// SIMATIC S7-200 project (STEP 7-Micro/WIN), CPU 224 CN REL 02.01

SYMBOL_TABLE USER1
P0_Reposo        M0.0     // Estado de espera inicial
P1_Sujecion      M0.1     // Estado de sujecion de la columna
P2_Empuje        M0.2     // Estado de entrega de la pieza inferior
P3_Retorno_E     M0.3     // Estado de retorno del cilindro de empuje
P4_Retorno_S     M0.4     // Estado de liberacion de la columna
T0_Inicio        M1.0     // Transicion Inicio Ciclo
T1_Sujeto        M1.1     // Transicion Sujecion OK
T2_Entregado     M1.2     // Transicion Entrega OK
T3_Emp_Ret       M1.3     // Transicion Empuje Retraido
T4_Suj_Ret       M1.4     // Transicion Sujecion Retraida
Ev_Marcha        M2.0     // Evento Marcha presionado y Seta OK
Ev_Pieza         M2.1     // Evento Pieza en base detectada
Ev_CilP_Ext      M2.2     // Evento Cilindro pequeno extendido
Ev_CilL_Ext      M2.3     // Evento Cilindro largo extendido
Ev_CilL_Ret      M2.4     // Evento Cilindro largo retraido
Ev_CilP_Ret      M2.5     // Evento Cilindro pequeno retraido
Ev_Pos_Pieza     M2.6     // Evento pieza en posicion
Cil_Peq_Ext      I0.0     // Sensor cilindro pequeno extendido
Cil_Peq_Ret      I0.1     // Sensor cilindro pequeno retraido
Cil_Lrg_Ext      I0.2     // Sensor cilindro largo extendido
Cil_Lrg_Ret      I0.3     // Sensor cilindro largo retraido
Pos_Pieza        I0.4     // Sensor fotoelectrico posicion pieza
Presencia_Sup    I0.5     // Sensor presencia superior
Presencia_Inf    I0.6     // Sensor presencia inferior
Sensor_Induc     I0.7     // Sensor inductivo material metalico
Btn_Marcha       I1.2     // Pulsador verde de marcha
Btn_Paro         I1.3     // Pulsador rojo de paro
Seta_Emerg       I1.4     // Zeta de emergencia (NC)
Selector_Rot     I1.5     // Selector rotatorio
V_Cil_Peq        Q0.0     // Valvula cilindro pequeno
V_Cil_Lrg        Q0.1     // Valvula cilindro largo
Lamp_Amarilla    Q0.7     // Lampara de advertencia
Lamp_Verde       Q1.0     // Lampara de marcha
Lamp_Roja        Q1.1     // Lampara de paro o falla
Sol_AP           V0.0     // Solicitud Alimentacion a Procesamiento
Ack_Sol_AP       V1.0     // Reconocimiento AP
Ack_MA           V0.1     // Reconocimiento marcha Unidad de Alimentacion
Marcha_A         V1.1     // Solicitud de marcha para la Unidad de Alimentacion
Alim_OK          V0.2     // Unidad de Alimentacion disponible
END_SYMBOL_TABLE

SYMBOL_TABLE S7-200 Symbols
First_Scan_On    SM0.1    // 仅第一个扫描周期中接通为 ON
END_SYMBOL_TABLE

ORGANIZATION_BLOCK MAIN:OB1
TITLE=UNIDAD DE ALIMENTACION - RED DE PETRI (CIPN) - 5 MODULOS (V4)
//  LOGICA BASADA EN REDES DE PETRI INTERPRETADAS
//  MODULO 1: INICIALIZACION
//  MODULO 2: EVENTOS
//  MODULO 3: DISPARO
//  MODULO 4: DINAMICA
//  MODULO 5: ACCIONES
BEGIN
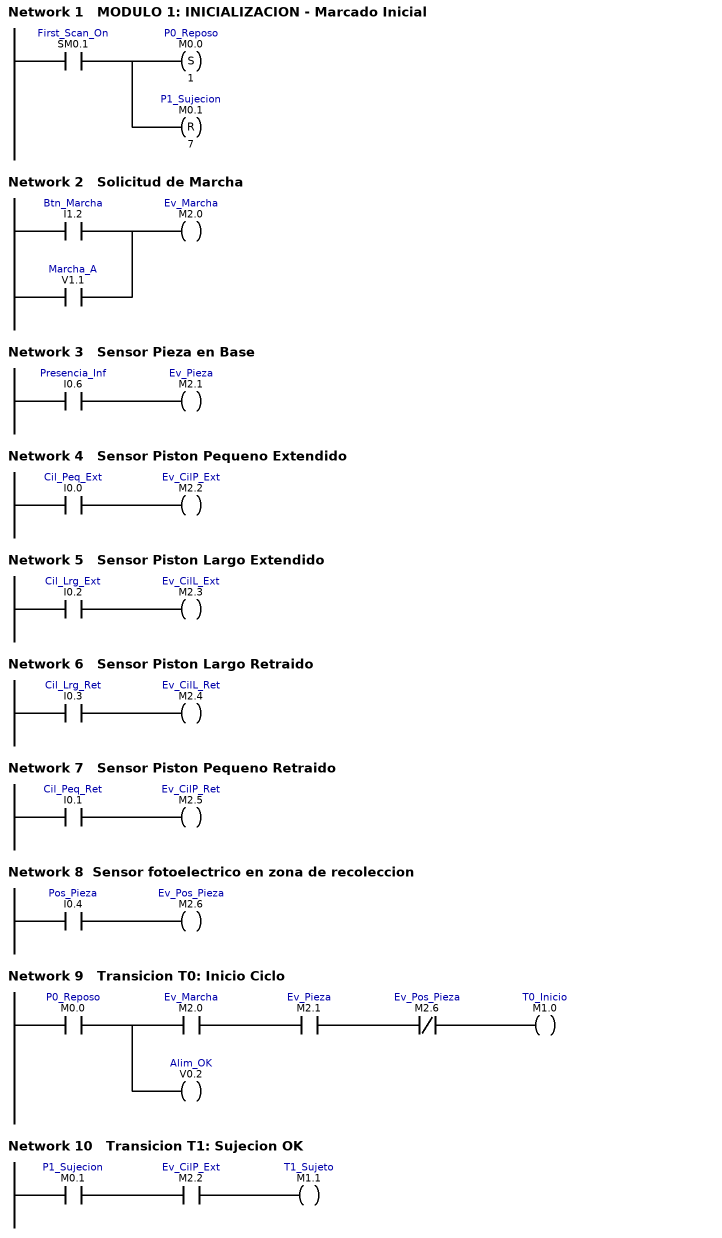
Network 1 //  MODULO 1: INICIALIZACION - Marcado Inicial
// P0 Reposo activo
// Limpieza de marcas P1-M0.7
// MODULO 2: EVENTOS (CAPTURA DE SENSORES)
LD     First_Scan_On:SM0.1
S      P0_Reposo:M0.0, 1
R      P1_Sujecion:M0.1, 7
Network 2 //  Solicitud de Marcha
LD     Btn_Marcha:I1.2
O      Marcha_A:V1.1
=      Ev_Marcha:M2.0
Network 3 //  Sensor Pieza en Base
LD     Presencia_Inf:I0.6
=      Ev_Pieza:M2.1
Network 4 //  Sensor Piston Pequeno Extendido
LD     Cil_Peq_Ext:I0.0
=      Ev_CilP_Ext:M2.2
Network 5 //  Sensor Piston Largo Extendido
LD     Cil_Lrg_Ext:I0.2
=      Ev_CilL_Ext:M2.3
Network 6 //  Sensor Piston Largo Retraido
LD     Cil_Lrg_Ret:I0.3
=      Ev_CilL_Ret:M2.4
Network 7 //  Sensor Piston Pequeno Retraido
// MODULO 3: CONDICIONES DE DISPARO (FIRING)
LD     Cil_Peq_Ret:I0.1
=      Ev_CilP_Ret:M2.5
Network 8 // Sensor fotoelectrico en zona de recoleccion
LD     Pos_Pieza:I0.4
=      Ev_Pos_Pieza:M2.6
Network 9 //  Transicion T0: Inicio Ciclo
LD     P0_Reposo:M0.0
LPS
A      Ev_Marcha:M2.0
A      Ev_Pieza:M2.1
AN     Ev_Pos_Pieza:M2.6
=      T0_Inicio:M1.0
LPP
=      Alim_OK:V0.2
Network 10 //  Transicion T1: Sujecion OK
LD     P1_Sujecion:M0.1
A      Ev_CilP_Ext:M2.2
=      T1_Sujeto:M1.1
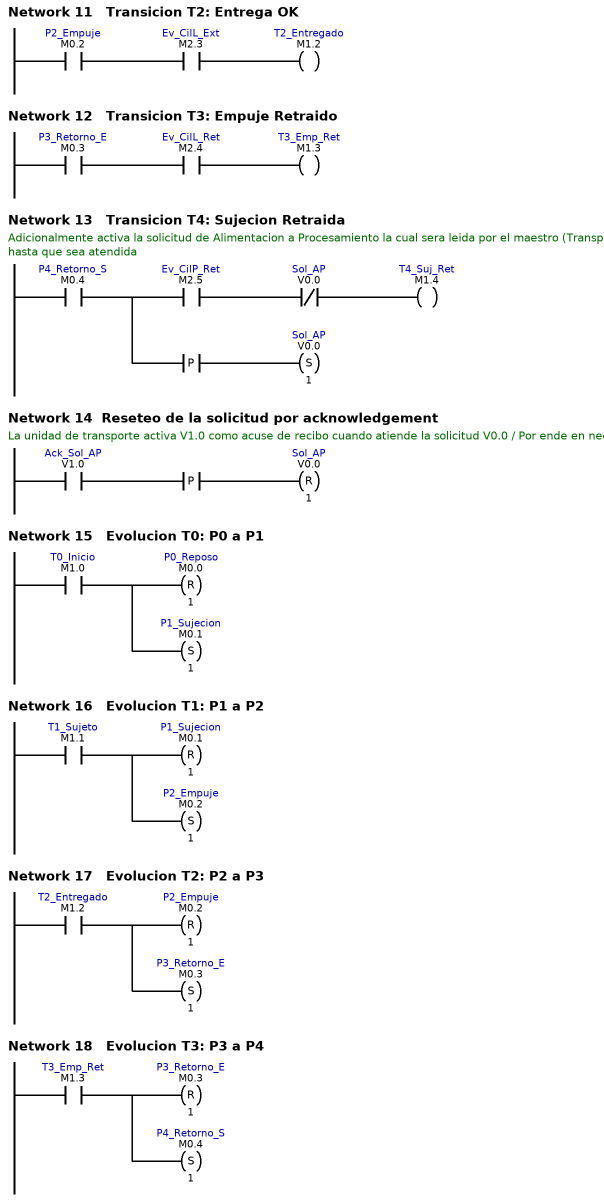
Network 11 //  Transicion T2: Entrega OK
LD     P2_Empuje:M0.2
A      Ev_CilL_Ext:M2.3
=      T2_Entregado:M1.2
Network 12 //  Transicion T3: Empuje Retraido
LD     P3_Retorno_E:M0.3
A      Ev_CilL_Ret:M2.4
=      T3_Emp_Ret:M1.3
Network 13 //  Transicion T4: Sujecion Retraida
// Adicionalmente activa la solicitud de Alimentacion a Procesamiento la cual sera leida por el maestro (Transporte)
// Esta solicitud funciona como enclavamiento que impide volver al estado de reposo hasta que sea atendida
// MODULO 4: DINAMICA DE LA RED (EVOLUCION DE ESTADOS)
LD     P4_Retorno_S:M0.4
LPS
A      Ev_CilP_Ret:M2.5
AN     Sol_AP:V0.0
=      T4_Suj_Ret:M1.4
LPP
EU
S      Sol_AP:V0.0, 1
Network 14 // Reseteo de la solicitud por acknowledgement
// La unidad de transporte activa V1.0 como acuse de recibo cuando atiende la solicitud V0.0
// Por ende en necesario desactivar la solicitud para evitar repeticiones.
LD     Ack_Sol_AP:V1.0
EU
R      Sol_AP:V0.0, 1
Network 15 //  Evolucion T0: P0 a P1
LD     T0_Inicio:M1.0
R      P0_Reposo:M0.0, 1
S      P1_Sujecion:M0.1, 1
Network 16 //  Evolucion T1: P1 a P2
LD     T1_Sujeto:M1.1
R      P1_Sujecion:M0.1, 1
S      P2_Empuje:M0.2, 1
Network 17 //  Evolucion T2: P2 a P3
LD     T2_Entregado:M1.2
R      P2_Empuje:M0.2, 1
S      P3_Retorno_E:M0.3, 1
Network 18 //  Evolucion T3: P3 a P4
LD     T3_Emp_Ret:M1.3
R      P3_Retorno_E:M0.3, 1
S      P4_Retorno_S:M0.4, 1
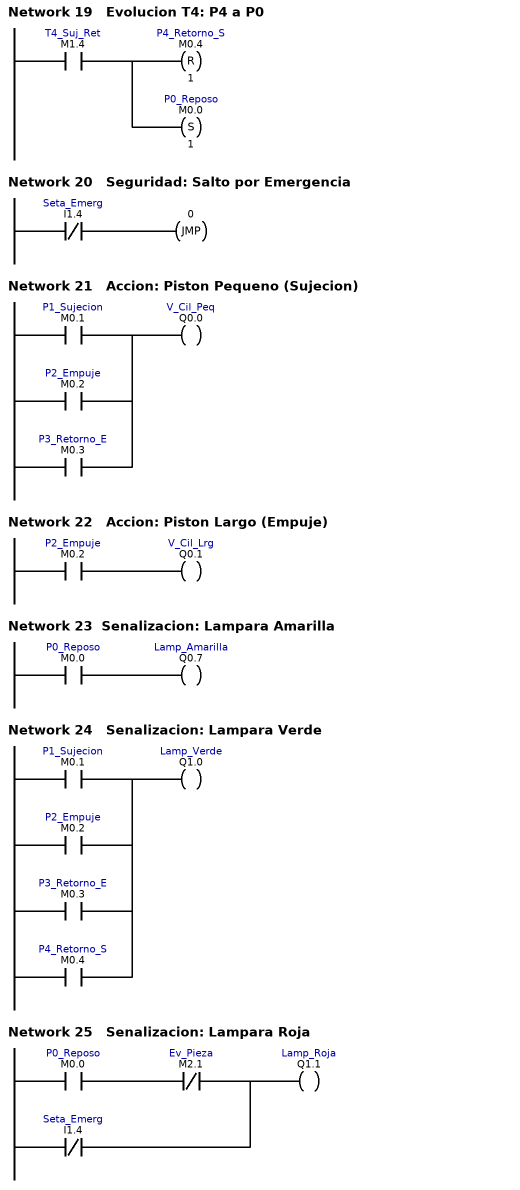
Network 19 //  Evolucion T4: P4 a P0
LD     T4_Suj_Ret:M1.4
R      P4_Retorno_S:M0.4, 1
S      P0_Reposo:M0.0, 1
Network 20 //  Seguridad: Salto por Emergencia
// MODULO 5: ACCIONES (SALIDAS FISICAS)
LDN    Seta_Emerg:I1.4
JMP    0
Network 21 //  Accion: Piston Pequeno (Sujecion)
LD     P1_Sujecion:M0.1
O      P2_Empuje:M0.2
O      P3_Retorno_E:M0.3
=      V_Cil_Peq:Q0.0
Network 22 //  Accion: Piston Largo (Empuje)
LD     P2_Empuje:M0.2
=      V_Cil_Lrg:Q0.1
Network 23 // Senalizacion: Lampara Amarilla	
LD     P0_Reposo:M0.0
=      Lamp_Amarilla:Q0.7
Network 24 //  Senalizacion: Lampara Verde
LD     P1_Sujecion:M0.1
O      P2_Empuje:M0.2
O      P3_Retorno_E:M0.3
O      P4_Retorno_S:M0.4
=      Lamp_Verde:Q1.0
Network 25 //  Senalizacion: Lampara Roja
LD     P0_Reposo:M0.0
AN     Ev_Pieza:M2.1
ON     Seta_Emerg:I1.4
=      Lamp_Roja:Q1.1
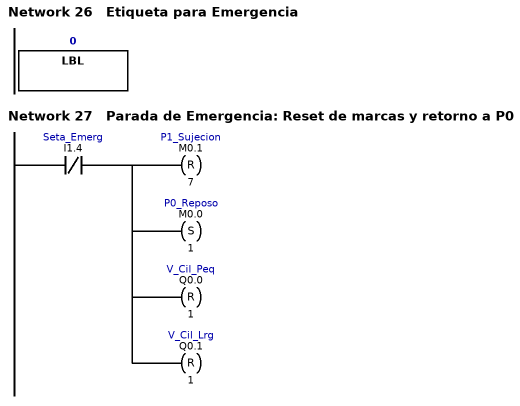
Network 26 //  Etiqueta para Emergencia
LBL    0
Network 27 //  Parada de Emergencia: Reset de marcas y retorno a P0
LDN    Seta_Emerg:I1.4
R      P1_Sujecion:M0.1, 7
S      P0_Reposo:M0.0, 1
R      V_Cil_Peq:Q0.0, 1
R      V_Cil_Lrg:Q0.1, 1
END_ORGANIZATION_BLOCK
